FUNCTION_BLOCK SM_Palletizer EXTENDS StateMachine
VAR_INPUT
	bExecute : BOOL;
	scFirstFloor : SC_FirstFloor;	
	scSecondFloor : SC_SecondFloor;
END_VAR
VAR_IN_OUT
	ioChainController : FB_ChainController;
END_VAR
VAR_OUTPUT
	
	bAllPartsPresent: BOOL;	
	
END_VAR
VAR

	fbDoneCycle : BoolOut;
	fbStepWorkerBusy : FB_StepWorker;
	
	
END_VAR

SUPER^();
scFirstFloor(bExecute := bExecute);
scSecondFloor(bExecute := bExecute);

bAllPartsPresent := scSecondFloor.bAllPartsPresent;
scSecondFloor.bPlateOpen := scFirstFloor.bPlateOpen;

METHOD PROTECTED   Busy : BOOL
VAR_INPUT
END_VAR
scFirstFloor(bExecute := TRUE);
scSecondFloor(bExecute := TRUE);
END_METHOD

METHOD PROTECTED  Error : BOOL
VAR_INPUT
END_VAR
END_METHOD

PROPERTY getDoneCycle : I_StepCondition
GET
getDoneCycle := fbDoneCycle;
END_GET
END_PROPERTY

METHOD PROTECTED  Idle : BOOL
VAR_INPUT
END_VAR
Start();
END_METHOD

METHOD PROTECTED  Init : BOOL
VAR_INPUT
END_VAR
ioChainController
	.addChain(itfChain := scFirstFloor)
	.addChain(itfChain := scSecondFloor);
	
scFirstFloor(
	sChainName := 'scFirstFloor',
	rChainController := ioChainController
);
scSecondFloor(
	sChainName := 'scSecondFloor',
	rChainController := ioChainController
);
Start();
END_METHOD

METHOD PROTECTED  Prepare : BOOL
VAR_INPUT
END_VAR
END_METHOD

METHOD PROTECTED  Ready : BOOL
VAR_INPUT
END_VAR
END_METHOD

METHOD PROTECTED  Waiting : BOOL
VAR_INPUT
END_VAR
END_METHOD

END_FUNCTION_BLOCK

(* stored: Version 1.1.0.1, ProductVersion 3.1.4024.2
   POU SM_Palletizer: Id {ce52986e-d795-4498-b449-1f0f8887e1e6}, SpecialFunc None
   Method Busy: Id {73f86d69-d2e5-4361-83bd-9fd09001ce81}
   Method Error: Id {0aa84eeb-c74a-4552-ae6d-56f85f508303}
   Property getDoneCycle: Id {da487bee-2a85-42f6-8ecb-c34e2f815fad}
   Get Get: Id {b3b5795f-92ac-48f0-b2da-b92918c7358d}
   Method Idle: Id {e02fc5be-2003-4821-a34b-ebb230a9eb31}
   Method Init: Id {a7562592-ad57-424e-8965-d7b38793483f}
   Method Prepare: Id {5e41363b-2ef9-4a2e-a5fa-7da58e2da2bc}
   Method Ready: Id {6aeac2e6-dd92-4451-b62a-3dd9ffa72f06}
   Method Waiting: Id {acd9be17-1066-42d2-ac59-aefa5bb57858} *)
